		30:
			ActualResult := TestFBBusy.Busy;
			AssertEquals_BOOL(Expected := ExpectedResult, Actual := ActualResult, Message := 'Function Block was not busy when Extending');
			TEST_FINISHED();
			State := State + 10;
	END_CASE

	//Call to FB Cyclic Logic
	TestFBBusy.CyclicLogic();
END_IF
END_METHOD

METHOD CommandInhibited
VAR_INST
	State		   : INT;
	ActualResult   : BOOL;
	ExpectedResult : BOOL := TRUE;
END_VAR
IF TEST_ORDERED('CommandInhibitedAlarm') THEN
	CASE State OF
		0:
			IF TestFBAlarm15.InitComplete THEN
				TestFBAlarm15.Override := 0;
				TestFBAlarm15.MoveAbsolute(100, TRUE);
				State := State + 10;
			END_IF

		10:
			IF TestFBAlarm15.Error OR (TestFBAlarm15.InPosition AND NOT TestFBAlarm15.Busy) THEN
				ActualResult := TestFBAlarm15.BasicAxisAlarms[E_BasicAxis.CommandWhileInhibited].bRaised;
				State		 := State + 10;
			END_IF

		20:
			AssertEquals_BOOL(Expected := ExpectedResult, Actual := ActualResult, Message := 'The alarm was not raised for Command Inhibited Error');
			TEST_FINISHED();
			State := State + 10;
	END_CASE

	TestFBAlarm15.CyclicLogic();
END_IF
END_METHOD

METHOD Init
VAR_INST
	State		   : INT;
	ActualResult   : BOOL;
	ExpectedResult : BOOL := TRUE;
	Timeout		   : TON;
END_VAR
IF TEST_ORDERED('BasicAxisInit') THEN
	CASE State OF
		0:
			Timeout.IN := TRUE;
			State	   := State + 10;

		10:
			IF TestFBInit.InitComplete AND NOT TestFBInit.Busy THEN
				State := State + 10;
			END_IF

			IF Timeout.Q THEN
				State := State + 10;
			END_IF

		20:
			ActualResult := TestFBInit.InitComplete;
			AssertEquals_BOOL(Expected := ExpectedResult, Actual := ActualResult, Message := 'Function Block did not init complete in 2s');
			TEST_FINISHED();
			State := State + 10;
	END_CASE

	//Call to FB Cyclic Logic
	Timeout(PT := T#2S);
	TestFBInit.CyclicLogic();
END_IF
END_METHOD

METHOD MCHaltAlarm
VAR_INST
	State		   : INT;
	ActualResult   : BOOL;
	ExpectedResult : BOOL := TRUE;
	WriteADS	   : FB_WriteAdsSymByName;
END_VAR
IF TEST_ORDERED('MCHaltAlarm') THEN
	CASE State OF
		0:
			WriteADS(bWrite	  := TRUE,
					 sNetId	  := '',
					 nPort	  := 851,
					 sVarName := 'PRG_TEST.ComponentBasicAxisTest.TestFBAlarm4.BasicAxis.MCHalt.Error',
					 nSrcAddr := ADR(ExpectedResult),
					 nLen	  := SIZEOF(ExpectedResult),
					 tTimeout := T#2S,
					 eComMode :=,
					 bBusy	  =>,
					 bError	  =>,
					 nErrorId =>);

			IF NOT WriteADS.bBusy OR WriteADS.bError THEN
				State := State + 10;
			END_IF

			IF TestFBAlarm4.BasicAxisAlarms[E_BasicAxis.HaltError].bRaised THEN
				ActualResult := TestFBAlarm4.BasicAxisAlarms[E_BasicAxis.HaltError].bRaised;
				State		 := State + 10;
			END_IF

		10:
			AssertEquals_BOOL(Expected := ExpectedResult, Actual := ActualResult, Message := 'The alarm was not raised for MC_Halt.Error');
			TEST_FINISHED();
			State := State + 10;
	END_CASE

	TestFBAlarm4.CyclicLogic();
END_IF
END_METHOD

METHOD MCHomeAlarm
VAR_INST
	State		   : INT;
	ActualResult   : BOOL;
	ExpectedResult : BOOL := TRUE;
	WriteADS	   : FB_WriteAdsSymByName;
END_VAR
IF TEST_ORDERED('MCHomeAlarm') THEN
	CASE State OF
		0:
			WriteADS(bWrite	  := TRUE,
					 sNetId	  := '',
					 nPort	  := 851,
					 sVarName := 'PRG_TEST.ComponentBasicAxisTest.TestFBAlarm6.BasicAxis.DefaultHome._Error',
					 nSrcAddr := ADR(ExpectedResult),
					 nLen	  := SIZEOF(ExpectedResult),
					 tTimeout := T#2S,
					 eComMode :=,
					 bBusy	  =>,
					 bError	  =>,
					 nErrorId =>);

			IF NOT WriteADS.bBusy OR WriteADS.bError THEN
				State := State + 10;
			END_IF

			IF TestFBAlarm6.BasicAxisAlarms[E_BasicAxis.HomeError].bRaised THEN
				ActualResult := TestFBAlarm6.BasicAxisAlarms[E_BasicAxis.HomeError].bRaised;
				State		 := State + 10;
			END_IF

		10:
			AssertEquals_BOOL(Expected := ExpectedResult, Actual := ActualResult, Message := 'The alarm was not raised for HomeMethod.Error');
			TEST_FINISHED();
			State := State + 10;
	END_CASE

	TestFBAlarm6.CyclicLogic();
END_IF
END_METHOD

METHOD MCJogAlarm
VAR_INST
	State		   : INT;
	ActualResult   : BOOL;
	ExpectedResult : BOOL := TRUE;
	WriteADS	   : FB_WriteAdsSymByName;
END_VAR
IF TEST_ORDERED('MCJogAlarm') THEN
	CASE State OF
		0:
			WriteADS(bWrite	  := TRUE,
					 sNetId	  := '',
					 nPort	  := 851,
					 sVarName := 'PRG_TEST.ComponentBasicAxisTest.TestFBAlarm7.BasicAxis.MCJog.Error',
					 nSrcAddr := ADR(ExpectedResult),
					 nLen	  := SIZEOF(ExpectedResult),
					 tTimeout := T#2S,
					 eComMode :=,
					 bBusy	  =>,
					 bError	  =>,
					 nErrorId =>);

			IF NOT WriteADS.bBusy OR WriteADS.bError THEN
				State := State + 10;
			END_IF

			IF TestFBAlarm7.BasicAxisAlarms[E_BasicAxis.JogError].bRaised THEN
				ActualResult := TestFBAlarm7.BasicAxisAlarms[E_BasicAxis.JogError].bRaised;
				State		 := State + 10;
			END_IF

		10:
			AssertEquals_BOOL(Expected := ExpectedResult, Actual := ActualResult, Message := 'The alarm was not raised for MCJog.Error');
			TEST_FINISHED();
			State := State + 10;
	END_CASE

	TestFBAlarm7.CyclicLogic();
END_IF
END_METHOD

METHOD MCMoveAbsoluteAlarm
VAR_INST
	State		   : INT;
	ActualResult   : BOOL;
	ExpectedResult : BOOL := TRUE;
END_VAR
IF TEST_ORDERED('MCMoveAbsAlarm') THEN
	CASE State OF
		0:
			IF TestFBAlarm8.InitComplete THEN
				TestFBAlarm8.MoveAbsolute(100, TRUE);
				State := State + 10;
			END_IF

		10:
			IF TestFBAlarm8.Error OR (TestFBAlarm8.InPosition AND NOT TestFBAlarm8.Busy) THEN
				State := State + 10;
			END_IF

		20:
			ActualResult := TestFBAlarm8.BasicAxisAlarms[E_BasicAxis.MoveAbsoluteError].bRaised;
			AssertEquals_BOOL(Expected := ExpectedResult, Actual := ActualResult, Message := 'The alarm was not raised for Move Absolute Error');
			TEST_FINISHED();
			State := State + 10;
	END_CASE

	TestFBAlarm8.CyclicLogic();
END_IF
END_METHOD

METHOD MCMoveModulo
VAR_INST
	State		   : INT;
	ActualResult   : BOOL;
	ExpectedResult : BOOL := TRUE;
END_VAR
IF TEST_ORDERED('MCMoveModuloAlarm') THEN
	CASE State OF
		0:
			IF TestFBAlarm11.InitComplete THEN
				TestFBAlarm11.MoveModulo(100, MC_Direction.MC_Positive_Direction, TRUE);
				State := State + 10;
			END_IF

		10:
			IF TestFBAlarm11.Error OR (TestFBAlarm11.InPosition AND NOT TestFBAlarm11.Busy) THEN
				State := State + 10;
			END_IF

		20:
			ActualResult := TestFBAlarm11.BasicAxisAlarms[E_BasicAxis.MoveModuloError].bRaised;
			AssertEquals_BOOL(Expected := ExpectedResult, Actual := ActualResult, Message := 'The alarm was not raised for Move Modulo Error');
			TEST_FINISHED();
			State := State + 10;
	END_CASE

	TestFBAlarm11.CyclicLogic();
END_IF
END_METHOD

METHOD MCMoveRelativeAlarm
VAR_INST
	State		   : INT;
	ActualResult   : BOOL;
	ExpectedResult : BOOL := TRUE;
END_VAR
IF TEST_ORDERED('MCMoveAbsAlarm') THEN
	CASE State OF
		0:
			IF TestFBAlarm9.InitComplete THEN
				TestFBAlarm9.MoveRelative(100, TRUE);
				State := State + 10;
			END_IF

		10:
			IF TestFBAlarm9.Error OR (TestFBAlarm9.InPosition AND NOT TestFBAlarm9.Busy) THEN
				State := State + 10;
			END_IF

		20:
			ActualResult := TestFBAlarm9.BasicAxisAlarms[E_BasicAxis.MoveRelativeError].bRaised;
			AssertEquals_BOOL(Expected := ExpectedResult, Actual := ActualResult, Message := 'The alarm was not raised for Move Relative Error');
			TEST_FINISHED();
			State := State + 10;
	END_CASE

	TestFBAlarm9.CyclicLogic();
END_IF
END_METHOD

METHOD MCMoveVelocity
VAR_INST
	State		   : INT;
	ActualResult   : BOOL;
	ExpectedResult : BOOL := TRUE;
END_VAR
IF TEST_ORDERED('MCMoveVelAlarm') THEN
	CASE State OF
		0:
			IF TestFBAlarm10.InitComplete THEN
				TestFBAlarm10.MoveVelocity(100, TRUE);
				State := State + 10;
			END_IF

		10:
			IF TestFBAlarm10.Error OR (TestFBAlarm10.InPosition AND NOT TestFBAlarm10.Busy) THEN
				State := State + 10;
			END_IF

		20:
			ActualResult := TestFBAlarm10.BasicAxisAlarms[E_BasicAxis.MoveVelocityError].bRaised;
			AssertEquals_BOOL(Expected := ExpectedResult, Actual := ActualResult, Message := 'The alarm was not raised for Move Relative Error');
			TEST_FINISHED();
			State := State + 10;
	END_CASE

	TestFBAlarm10.CyclicLogic();
END_IF
END_METHOD

METHOD MCPowerAlarm
VAR_INST
	State		   : INT;
	ActualResult   : BOOL;
	ExpectedResult : BOOL := TRUE;
	WriteADS	   : FB_WriteAdsSymByName;
END_VAR
IF TEST_ORDERED('MCPowerAlarm') THEN
	CASE State OF
		0:
			WriteADS(bWrite	  := TRUE,
					 sNetId	  := '',
					 nPort	  := 851,
					 sVarName := 'PRG_TEST.ComponentBasicAxisTest.TestFBAlarm2.BasicAxis.MCPower.Error',
					 nSrcAddr := ADR(ExpectedResult),
					 nLen	  := SIZEOF(ExpectedResult),
					 tTimeout := T#2S,
					 eComMode :=,
					 bBusy	  =>,
					 bError	  =>,
					 nErrorId =>);

			IF NOT WriteADS.bBusy OR WriteADS.bError THEN
				State := State + 10;
			END_IF

			IF TestFBAlarm2.BasicAxisAlarms[E_BasicAxis.PowerError].bRaised THEN
				ActualResult := TestFBAlarm2.BasicAxisAlarms[E_BasicAxis.PowerError].bRaised;
				State		 := State + 10;
			END_IF

		10:
			AssertEquals_BOOL(Expected := ExpectedResult, Actual := ActualResult, Message := 'The alarm was not raised for MC_Power.Error');
			TEST_FINISHED();
			State := State + 10;
	END_CASE

	TestFBAlarm2.CyclicLogic();
END_IF
END_METHOD

METHOD McReadAxisParametersAlarm
VAR_INST
	State		   : INT;
	ActualResult   : BOOL;
	ExpectedResult : BOOL := TRUE;
	WriteADS	   : FB_WriteAdsSymByName;
END_VAR
IF TEST_ORDERED('MCReadAxisAlarm') THEN
	CASE State OF
		0:
			WriteADS(bWrite	  := TRUE,
					 sNetId	  := '',
					 nPort	  := 851,
					 sVarName := 'PRG_TEST.ComponentBasicAxisTest.TestFBAlarm12.BasicAxis.MCReadParameterSet.Error',
					 nSrcAddr := ADR(ExpectedResult),
					 nLen	  := SIZEOF(ExpectedResult),
					 tTimeout := T#2S,
					 eComMode :=,
					 bBusy	  =>,
					 bError	  =>,
					 nErrorId =>);

			IF NOT WriteADS.bBusy OR WriteADS.bError THEN
				State := State + 10;
			END_IF

			IF TestFBAlarm12.BasicAxisAlarms[E_BasicAxis.ReadParameterSetError].bRaised THEN
				ActualResult := TestFBAlarm12.BasicAxisAlarms[E_BasicAxis.ReadParameterSetError].bRaised;
				State		 := State + 10;
			END_IF

		10:
			AssertEquals_BOOL(Expected := ExpectedResult, Actual := ActualResult, Message := 'The alarm was not raised for MC Read Axis Parameter Error');
			TEST_FINISHED();
			State := State + 10;
	END_CASE

	TestFBAlarm12.CyclicLogic();
END_IF
END_METHOD

METHOD MCResetAlarm
VAR_INST
	State		   : INT;
	ActualResult   : BOOL;
	ExpectedResult : BOOL := TRUE;
	WriteADS	   : FB_WriteAdsSymByName;
END_VAR
IF TEST_ORDERED('MCResetAlarm') THEN
	CASE State OF
		0:
			WriteADS(bWrite	  := TRUE,
					 sNetId	  := '',
					 nPort	  := 851,
					 sVarName := 'PRG_TEST.ComponentBasicAxisTest.TestFBAlarm3.BasicAxis.DefaultReset._Error',
					 nSrcAddr := ADR(ExpectedResult),
					 nLen	  := SIZEOF(ExpectedResult),
					 tTimeout := T#2S,
					 eComMode :=,
					 bBusy	  =>,
					 bError	  =>,
					 nErrorId =>);

			IF NOT WriteADS.bBusy OR WriteADS.bError THEN
				State := State + 10;
			END_IF

			IF TestFBAlarm3.BasicAxisAlarms[E_BasicAxis.ResetError].bRaised THEN
				ActualResult := TestFBAlarm3.BasicAxisAlarms[E_BasicAxis.ResetError].bRaised;
				State		 := State + 10;
			END_IF

		10:
			AssertEquals_BOOL(Expected := ExpectedResult, Actual := ActualResult, Message := 'The alarm was not raised for ResetMethod.Error');
			TEST_FINISHED();
			State := State + 10;
	END_CASE

	TestFBAlarm3.CyclicLogic();
END_IF
END_METHOD

METHOD McWriteAxisBoolParameterAlarm
VAR_INST
	State		   : INT;
	ActualResult   : BOOL;
	ExpectedResult : BOOL := TRUE;
	WriteADS	   : FB_WriteAdsSymByName;
END_VAR
IF TEST_ORDERED('MCWriteAxisBoolAlarm') THEN
	CASE State OF
		0:
			WriteADS(bWrite	  := TRUE,
					 sNetId	  := '',
					 nPort	  := 851,
					 sVarName := 'PRG_TEST.ComponentBasicAxisTest.TestFBAlarm14.BasicAxis.MCWriteBoolParameter.Error',
					 nSrcAddr := ADR(ExpectedResult),
					 nLen	  := SIZEOF(ExpectedResult),
					 tTimeout := T#2S,
					 eComMode :=,
					 bBusy	  =>,
					 bError	  =>,
					 nErrorId =>);

			IF NOT WriteADS.bBusy OR WriteADS.bError THEN
				State := State + 10;
			END_IF

			IF TestFBAlarm14.BasicAxisAlarms[E_BasicAxis.WriteBoolParameterError].bRaised THEN
				ActualResult := TestFBAlarm14.BasicAxisAlarms[E_BasicAxis.WriteBoolParameterError].bRaised;
				State		 := State + 10;
			END_IF

		10:
			AssertEquals_BOOL(Expected := ExpectedResult, Actual := ActualResult, Message := 'The alarm was not raised for MC Write Axis Bool Parameter Error');
			TEST_FINISHED();
			State := State + 10;
	END_CASE

	TestFBAlarm14.CyclicLogic();
END_IF
END_METHOD

METHOD McWriteAxisParameterAlarm
VAR_INST
	State		   : INT;
	ActualResult   : BOOL;
	ExpectedResult : BOOL := TRUE;
	WriteADS	   : FB_WriteAdsSymByName;
END_VAR
IF TEST_ORDERED('MCWriteAxisAlarm') THEN
	CASE State OF
		0:
			WriteADS(bWrite	  := TRUE,
					 sNetId	  := '',
					 nPort	  := 851,
					 sVarName := 'PRG_TEST.ComponentBasicAxisTest.TestFBAlarm13.BasicAxis.MCWriteParameter.Error',
					 nSrcAddr := ADR(ExpectedResult),
					 nLen	  := SIZEOF(ExpectedResult),
					 tTimeout := T#2S,
					 eComMode :=,
					 bBusy	  =>,
					 bError	  =>,
					 nErrorId =>);

			IF NOT WriteADS.bBusy OR WriteADS.bError THEN
				State := State + 10;
			END_IF

			IF TestFBAlarm13.BasicAxisAlarms[E_BasicAxis.WriteParameterError].bRaised THEN
				ActualResult := TestFBAlarm13.BasicAxisAlarms[E_BasicAxis.WriteParameterError].bRaised;
				State		 := State + 10;
			END_IF

		10:
			AssertEquals_BOOL(Expected := ExpectedResult, Actual := ActualResult, Message := 'The alarm was not raised for MC Write Axis Parameter Error');
			TEST_FINISHED();
			State := State + 10;
	END_CASE

	TestFBAlarm13.CyclicLogic();
END_IF
END_METHOD

METHOD NameSetProperty
VAR_INST
	State			: INT;
	ActualResult	: STRING;
	ActualResultHMI : STRING;
	ExpectedResult	: STRING := 'TEST_NAME';
END_VAR
IF TEST_ORDERED('BasicAxisNameSetProperty') THEN
	CASE State OF
		0:
			State := State + 10;

		10:
			IF TestFBNameSetProperty.InitComplete AND NOT TestFBNameSetProperty.Busy THEN
				State := State + 10;
			END_IF

		20:
			TestFBNameSetProperty.Name := ExpectedResult;
			State					   := State + 10;

		30:
			ActualResultHMI := TestFBNameSetProperty.ComponentBase_HMI.Config.Name;
			ActualResult	:= TestFBNameSetProperty.Name;
			AssertEquals(Expected := ExpectedResult, Actual := ActualResult, Message := 'Name was not read by Property correctly');
			AssertEquals(Expected := ExpectedResult, Actual := ActualResultHMI, Message := 'Name was not read by HMI correctly');
			TEST_FINISHED();
			State := State + 10;
	END_CASE

	//Call to FB Cyclic Logic
	TestFBNameSetProperty.CyclicLogic();
END_IF
END_METHOD

METHOD SimulationCheckAlarm
VAR_INST
	State		   : INT;
	ActualResult   : BOOL;
	ExpectedResult : BOOL := TRUE;
END_VAR
IF TEST_ORDERED('BasicAxisSimulationCheckAlarm') THEN
	CASE State OF
		0:
			State := State + 10;

		10:
			IF TestFBSimulationCheckAlarm.InitComplete AND NOT TestFBSimulationCheckAlarm.Busy THEN
				State := State + 10;
			END_IF

		20:
			TestFBSimulationCheckAlarm.InSimulation := TRUE; //Set simulation to true;
			State									:= State + 10;

		30:
			ActualResult := TestFBSimulationCheckAlarm.ComponentBaseAlarms[E_ComponentBase.SimulationWarning].bRaised;
			AssertEquals_BOOL(Expected := ExpectedResult, Actual := ActualResult, Message := 'Function Block did Raise alarm when in simulation');
			TEST_FINISHED();
			State := State + 10;
	END_CASE

	//Call to FB Cyclic Logic
	TestFBSimulationCheckAlarm.CyclicLogic();
END_IF
END_METHOD

METHOD SimulationSetHMI
VAR_INST
	State			: INT;
	ActualResult	: BOOL;
	ActualResultHMI : BOOL;
	ExpectedResult	: BOOL := TRUE;
	WriteADS		: FB_WriteAdsSymByName;
END_VAR
IF TEST_ORDERED('BasicAxisSetSimulationHMI') THEN
	CASE State OF
		0:
			State := State + 10;

		10:
			IF TestFBSimulationSetHMI.InitComplete AND NOT TestFBSimulationSetHMI.Busy THEN
				TestFBSimulationSetHMI.AllowHMIControl(); // Must turn on Allow control for code to function
				State := State + 10;
			END_IF

		20:
			WriteADS(bWrite	  := TRUE,
					 sNetId	  := '',
					 nPort	  := 851,
					 sVarName := 'PRG_TEST.ComponentBasicAxisTest.TestFBSimulationSetHMI.ComponentBase_HMI.Command.SimulatedOperation',
					 nSrcAddr := ADR(ExpectedResult),
					 nLen	  := SIZEOF(ExpectedResult),
					 tTimeout := T#2S,
					 eComMode :=,
					 bBusy	  =>,
					 bError	  =>,
					 nErrorId =>);

			IF NOT WriteADS.bBusy OR WriteADS.bError THEN
				State := State + 10;
			END_IF

		30:
			ActualResult	:= TestFBSimulationSetHMI.InSimulation;
			ActualResultHMI := TestFBSimulationSetHMI.ComponentBase_HMI.Status.InSimulation;
			AssertEquals_BOOL(Expected := ExpectedResult, Actual := ActualResult, Message := 'Function Block did not set simulation by HMI when read by Property');
			AssertEquals_BOOL(Expected := ExpectedResult, Actual := ActualResultHMI, Message := 'Function Block did not set simulation by HMI when read by HMI');
			TEST_FINISHED();
			State := State + 10;
	END_CASE

	//Call to FB Cyclic Logic
	TestFBSimulationSetHMI.CyclicLogic();
END_IF
END_METHOD

METHOD SimulationSetProperty
VAR_INST
	State			: INT;
	ActualResult	: BOOL;
	ActualResultHMI : BOOL;
	ExpectedResult	: BOOL := TRUE;
END_VAR
IF TEST_ORDERED('BasicAxisSetSimulationProperty') THEN
	CASE State OF
		0:
			State := State + 10;

		10:
			IF TestFBSimulationSetProperty.InitComplete AND NOT TestFBSimulationSetProperty.Busy THEN
				State := State + 10;
			END_IF

		20:
			TestFBSimulationSetProperty.InSimulation := TRUE;
			State									 := State + 10;

		30:
			ActualResult	:= TestFBSimulationSetProperty.InSimulation;
			ActualResultHMI := TestFBSimulationSetProperty.ComponentBase_HMI.Status.InSimulation;
			AssertEquals_BOOL(Expected := ExpectedResult, Actual := ActualResult, Message := 'Function Block did not set simulation by property when read by Property');
			AssertEquals_BOOL(Expected := ExpectedResult, Actual := ActualResultHMI, Message := 'Function Block did not set simulation by property when read by HMI');
			TEST_FINISHED();
			State := State + 10;
	END_CASE

	//Call to FB Cyclic Logic
	TestFBSimulationSetProperty.CyclicLogic();
END_IF
END_METHOD

END_FUNCTION_BLOCK

// Testing/PRG_TEST
PROGRAM PRG_TEST
VAR
	SingleSolenoidTest		   : FB_SingleSolenoid_Test;
	DoubleSolenoidTest		   : FB_DoubleSolenoid_Test;
	SingleSolenoidFeedbackTest : FB_SingleSolenoidFeedback_Test;
	ComponentBasicAxisTest	   : FB_ComponentBasicAxis_Test;
END_VAR

TcUnit.RUN();

END_PROGRAM

// Testing/Solenoids/FB_SingleSolenoid_Test
FUNCTION_BLOCK FB_SingleSolenoid_Test EXTENDS TcUnit.FB_TestSuite
VAR
	// FBs for ComponentBase
	TestFBInit					: FB_SingleSolenoid;
	TestFBNameSetProperty		: FB_SingleSolenoid;
	TestFBNameSetHMI			: FB_SingleSolenoid;
	TestFBSimulationSetProperty : FB_SingleSolenoid;
	TestFBSimulationSetHMI		: FB_SingleSolenoid;
	TestFBSimulationCheckAlarm	: FB_SingleSolenoid;
	TestFBBusy					: FB_SingleSolenoid;
	TestFBAllowHMI				: FB_SingleSolenoid;
	TestFBBlockHMI				: FB_SingleSolenoid;

	// Solenoid FB	
	TestSingleSolenoidExtend  : FB_SingleSolenoid;
	TestSingleSolenoidRetract : FB_SingleSolenoid;
END_VAR

Init();
NameSetProperty();
SimulationSetProperty();
SimulationSetHMI();
SimulationCheckAlarm();
Busy();
AllowHMI();
BlockHMI();
ExtendEqualsExtendedOutputOn();
RetractEqualsExtendOutputOff();

METHOD AllowHMI
VAR_INST
	State		   : INT;
	ActualResult   : BOOL;
	ExpectedResult : BOOL := TRUE;
END_VAR
IF TEST_ORDERED('AllowHMI') THEN
	CASE State OF
		0:
			State := State + 10;

		10:
			IF TestFBAllowHMI.InitComplete AND NOT TestFBAllowHMI.Busy THEN
				TestFBAllowHMI.AllowHMIControl();
				State := State + 10;
			END_IF

		20:
			ActualResult := TestFBAllowHMI.ComponentBase_HMI.Status.HMIControlAvailable;
			AssertEquals_BOOL(Expected := ExpectedResult, Actual := ActualResult, Message := 'Function Block read allow HMI Control in HMI Tag not true');
			TEST_FINISHED();
			State := State + 10;
	END_CASE

	//Call to FB Cyclic Logic
	TestFBAllowHMI.CyclicLogic();
END_IF
END_METHOD

METHOD BlockHMI
VAR_INST
	State		   : INT;
	ActualResult   : BOOL;
	ExpectedResult : BOOL := FALSE;
END_VAR
IF TEST_ORDERED('BlockHMI') THEN
	CASE State OF
		0:
			State := State + 10;

		10:
			IF TestFBBlockHMI.InitComplete AND NOT TestFBBlockHMI.Busy THEN
				TestFBBlockHMI.AllowHMIControl();
				State := State + 10;
			END_IF

		20:
			IF TestFBBlockHMI.ComponentBase_HMI.Status.HMIControlAvailable THEN
				TestFBBlockHMI.BlockHMIControl();
				State := State + 10;
			END_IF

		30:
			ActualResult := TestFBBlockHMI.ComponentBase_HMI.Status.HMIControlAvailable;
			AssertEquals_BOOL(Expected := ExpectedResult, Actual := ActualResult, Message := 'Function Block read Block HMI Control in HMI Tag not false');
			TEST_FINISHED();
			State := State + 10;
	END_CASE

	//Call to FB Cyclic Logic
	TestFBBlockHMI.CyclicLogic();
END_IF
END_METHOD

METHOD Busy
VAR_INST
	State		   : INT;
	ActualResult   : BOOL;
	ExpectedResult : BOOL := TRUE;
	Timeout		   : TON;
END_VAR
IF TEST_ORDERED('Busy') THEN
	CASE State OF
		0:
			State := State + 10;

		10:
			IF TestFBBusy.InitComplete AND NOT TestFBBusy.Busy THEN
				State := State + 10;
			END_IF

		20:
			TestFBBusy.Extend();
			State := State + 10;

		30:
			ActualResult := TestFBBusy.Busy;
			AssertEquals_BOOL(Expected := ExpectedResult, Actual := ActualResult, Message := 'Function Block was not busy when Extending');
			TEST_FINISHED();
			State := State + 10;
	END_CASE

	//Call to FB Cyclic Logic
	TestFBBusy.CyclicLogic();
END_IF
END_METHOD

METHOD ExtendEqualsExtendedOutputOn
VAR_INST
	State		   : INT;
	ActualResult   : BOOL;
	ExpectedResult : BOOL := TRUE;
END_VAR
IF TEST_ORDERED('ExtendEqualsExtendedOutputOn') THEN
	CASE State OF
		0:
			State := State + 10;

		10:
			TestSingleSolenoidExtend.Extend();
			State := State + 10;

		20:
			ActualResult := TestSingleSolenoidExtend.ExtendOutput;
			AssertEquals_BOOL(Expected := ExpectedResult, Actual := ActualResult, Message := 'Solenoid did not set output on');
			TEST_FINISHED();
			State := State + 10;
	END_CASE

	TestSingleSolenoidExtend.CyclicLogic();
END_IF
END_METHOD

METHOD Init
VAR_INST
	State		   : INT;
	ActualResult   : BOOL;
	ExpectedResult : BOOL := TRUE;
	Timeout		   : TON;
END_VAR
IF TEST_ORDERED('Init') THEN
	CASE State OF
		0:
			Timeout.IN := TRUE;
			State	   := State + 10;

		10:
			IF TestFBInit.InitComplete AND NOT TestFBInit.Busy THEN
				State := State + 10;
			END_IF

			IF Timeout.Q THEN
				State := State + 10;
			END_IF

		20:
			ActualResult := TestFBInit.InitComplete;
			AssertEquals_BOOL(Expected := ExpectedResult, Actual := ActualResult, Message := 'Function Block did not init complete in 2s');
			TEST_FINISHED();
			State := State + 10;
	END_CASE

	//Call to FB Cyclic Logic
	Timeout(PT := T#2S);
	TestFBInit.CyclicLogic();
END_IF
END_METHOD

METHOD NameSetProperty
VAR_INST
	State			: INT;
	ActualResult	: STRING;
	ActualResultHMI : STRING;
	ExpectedResult	: STRING := 'TEST_NAME';
END_VAR
IF TEST_ORDERED('NameSetProperty') THEN
	CASE State OF
		0:
			State := State + 10;

		10:
			IF TestFBNameSetProperty.InitComplete AND NOT TestFBNameSetProperty.Busy THEN
				State := State + 10;
			END_IF

		20:
			TestFBNameSetProperty.Name := ExpectedResult;
			State					   := State + 10;

		30:
			ActualResultHMI := TestFBNameSetProperty.ComponentBase_HMI.Config.Name;
			ActualResult	:= TestFBNameSetProperty.Name;
			AssertEquals(Expected := ExpectedResult, Actual := ActualResult, Message := 'Name was not read by Property correctly');
			AssertEquals(Expected := ExpectedResult, Actual := ActualResultHMI, Message := 'Name was not read by HMI correctly');
			TEST_FINISHED();
			State := State + 10;
	END_CASE

	//Call to FB Cyclic Logic
	TestFBNameSetProperty.CyclicLogic();
END_IF
END_METHOD

METHOD RetractEqualsExtendOutputOff
VAR_INST
	State		   : INT;
	ActualResult   : BOOL;
	ExpectedResult : BOOL := FALSE;
END_VAR
IF TEST_ORDERED('RetractEqualsExtendOutputOff') THEN
	CASE State OF
		0:
			State := State + 10;

		10:
			TestSingleSolenoidRetract.Retract();
			State := State + 10;

		20:
			ActualResult := TestSingleSolenoidRetract.ExtendOutput;
			AssertEquals_BOOL(Expected := ExpectedResult, Actual := ActualResult, Message := 'Solenoid did not set output on');
			TEST_FINISHED();
			State := State + 10;
	END_CASE

	TestSingleSolenoidRetract.CyclicLogic();
END_IF
END_METHOD

METHOD SimulationCheckAlarm
VAR_INST
	State		   : INT;
	ActualResult   : BOOL;
	ExpectedResult : BOOL := TRUE;
END_VAR
IF TEST_ORDERED('SimulationCheckAlarm') THEN
	CASE State OF
		0:
			State := State + 10;

		10:
			IF TestFBSimulationCheckAlarm.InitComplete AND NOT TestFBSimulationCheckAlarm.Busy THEN
				State := State + 10;
			END_IF

		20:
			TestFBSimulationCheckAlarm.InSimulation := TRUE; //Set simulation to true;
			State									:= State + 10;

		30:
			ActualResult := TestFBSimulationCheckAlarm.ComponentBaseAlarms[E_ComponentBase.SimulationWarning].bRaised;
			AssertEquals_BOOL(Expected := ExpectedResult, Actual := ActualResult, Message := 'Function Block did Raise alarm when in simulation');
			TEST_FINISHED();
			State := State + 10;
	END_CASE

	//Call to FB Cyclic Logic
	TestFBSimulationCheckAlarm.CyclicLogic();
END_IF
END_METHOD

METHOD SimulationSetHMI
VAR_INST
	State			: INT;
	ActualResult	: BOOL;
	ActualResultHMI : BOOL;
	ExpectedResult	: BOOL := TRUE;
	WriteADS		: FB_WriteAdsSymByName;
END_VAR
IF TEST_ORDERED('SimulationSetHMI') THEN
	CASE State OF
		0:
			State := State + 10;

		10:
			IF TestFBSimulationSetHMI.InitComplete AND NOT TestFBSimulationSetHMI.Busy THEN
				TestFBSimulationSetHMI.AllowHMIControl(); // Must turn on Allow control for code to function
				State := State + 10;
			END_IF

		20:
			WriteADS(bWrite	  := TRUE,
					 sNetId	  := '',
					 nPort	  := 851,
					 sVarName := 'PRG_TEST.SingleSolenoidTest.TestFBSimulationSetHMI.ComponentBase_HMI.Command.SimulatedOperation',
					 nSrcAddr := ADR(ExpectedResult),
					 nLen	  := SIZEOF(ExpectedResult),
					 tTimeout := T#2S,
					 eComMode :=,
					 bBusy	  =>,
					 bError	  =>,
					 nErrorId =>);

			IF NOT WriteADS.bBusy OR WriteADS.bError THEN
				State := State + 10;
			END_IF

		30:
			ActualResult	:= TestFBSimulationSetHMI.InSimulation;
			ActualResultHMI := TestFBSimulationSetHMI.ComponentBase_HMI.Status.InSimulation;
			AssertEquals_BOOL(Expected := ExpectedResult, Actual := ActualResult, Message := 'Function Block did not set simulation by HMI when read by Property');
			AssertEquals_BOOL(Expected := ExpectedResult, Actual := ActualResultHMI, Message := 'Function Block did not set simulation by HMI when read by HMI');
			TEST_FINISHED();
			State := State + 10;
	END_CASE

	//Call to FB Cyclic Logic
	TestFBSimulationSetHMI.CyclicLogic();
END_IF
END_METHOD

METHOD SimulationSetProperty
VAR_INST
	State			: INT;
	ActualResult	: BOOL;
	ActualResultHMI : BOOL;
	ExpectedResult	: BOOL := TRUE;
END_VAR
IF TEST_ORDERED('SimulationSetProperty') THEN
	CASE State OF
		0:
			State := State + 10;

		10:
			IF TestFBSimulationSetProperty.InitComplete AND NOT TestFBSimulationSetProperty.Busy THEN
				State := State + 10;
			END_IF

		20:
			TestFBSimulationSetProperty.InSimulation := TRUE;
			State									 := State + 10;

		30:
			ActualResult	:= TestFBSimulationSetProperty.InSimulation;
			ActualResultHMI := TestFBSimulationSetProperty.ComponentBase_HMI.Status.InSimulation;
			AssertEquals_BOOL(Expected := ExpectedResult, Actual := ActualResult, Message := 'Function Block did not set simulation by property when read by Property');
			AssertEquals_BOOL(Expected := ExpectedResult, Actual := ActualResultHMI, Message := 'Function Block did not set simulation by property when read by HMI');
			TEST_FINISHED();
			State := State + 10;
	END_CASE

	//Call to FB Cyclic Logic
	TestFBSimulationSetProperty.CyclicLogic();
END_IF
END_METHOD

END_FUNCTION_BLOCK

// Testing/Solenoids/FB_DoubleSolenoid_Test
FUNCTION_BLOCK FB_DoubleSolenoid_Test EXTENDS TcUnit.FB_TestSuite
VAR
	TestFBExtend  : FB_DoubleSolenoid;
	TestFBRetract : FB_DoubleSolenoid;
END_VAR

ExtendEqualsExtendOutputOnRetractOff();
RetractEqualsExtendOutputOffRetractOutputOn();

METHOD ExtendEqualsExtendOutputOnRetractOff
VAR_INST
	State						: INT;
	ActualExtendOutputResult	: BOOL;
	ActualRetractOutputResult	: BOOL;
	ExpectedExtendOutputResult	: BOOL := TRUE;
	ExpectedRetractOutputResult : BOOL := FALSE;
END_VAR
IF TEST_ORDERED('ExtendEqualsExtendOutputOnRetractOff') THEN
	CASE State OF
		0:
			State := State + 10;

		10:
			IF TestFBExtend.InitComplete AND NOT TestFBExtend.Busy THEN
				TestFBExtend.Extend();
				State := State + 10;
			END_IF

		20:
			ActualExtendOutputResult := TestFBExtend.ExtendOutput;
			AssertEquals_BOOL(Expected := ExpectedExtendOutputResult, Actual := ActualExtendOutputResult, Message := 'Solenoid did not set extend output on');
			ActualRetractOutputResult := TestFBExtend.RetractOutput;
			AssertEquals_BOOL(Expected := ExpectedRetractOutputResult, Actual := ActualRetractOutputResult, Message := 'Solenoid did not set retract output off');
			TEST_FINISHED();
			State := State + 10;
	END_CASE

	TestFBExtend.CyclicLogic();
END_IF
END_METHOD

METHOD RetractEqualsExtendOutputOffRetractOutputOn
VAR_INST
	State						: INT;
	ActualExtendOutputResult	: BOOL;
	ActualRetractOutputResult	: BOOL;
	ExpectedExtendOutputResult	: BOOL := FALSE;
	ExpectedRetractOutputResult : BOOL := TRUE;
END_VAR
IF TEST_ORDERED('ExtendEqualsExtendOutputOffRetractOn') THEN
	CASE State OF
		0:
			State := State + 10;

		10:
			IF TestFBRetract.InitComplete AND NOT TestFBRetract.Busy THEN
				TestFBRetract.Extend();
				State := State + 10;
			END_IF

		20:
			IF TestFBRetract.Extended THEN
				TestFBRetract.Retract();
				State := State + 10;
			END_IF

		30:
			ActualExtendOutputResult := TestFBRetract.ExtendOutput;
			AssertEquals_BOOL(Expected := ExpectedExtendOutputResult, Actual := ActualExtendOutputResult, Message := 'Solenoid did not set extend output off');
			ActualRetractOutputResult := TestFBRetract.RetractOutput;
			AssertEquals_BOOL(Expected := ExpectedRetractOutputResult, Actual := ActualRetractOutputResult, Message := 'Solenoid did not set retract output on');
			TEST_FINISHED();
			State := State + 10;
	END_CASE

	TestFBRetract.CyclicLogic();
END_IF
END_METHOD

END_FUNCTION_BLOCK

// Testing/Solenoids/FB_SingleSolenoidFeedback_Test
FUNCTION_BLOCK FB_SingleSolenoidFeedback_Test EXTENDS FB_TestSuite
VAR
	// Solenoid FB	
	TestSingleSolenoidFeedbackExtend	   : FB_SingleSolenoidFeedback;
	TestSingleSolenoidFeedbackExtendError  : FB_SingleSolenoidFeedback;
	TestSingleSolenoidFeedbackRetract	   : FB_SingleSolenoidFeedback;
	TestSingleSolenoidFeedbackRetractError : FB_SingleSolenoidFeedback;
END_VAR

Extend();
ExtendError();

METHOD Extend
VAR_INST
	State		   : INT;
	ActualResult   : BOOL;
	ExpectedResult : BOOL := TRUE;
END_VAR
IF TEST_ORDERED('SingleSolenoidFeedbackTestExtend') THEN
	CASE State OF
		0:
			IF TestSingleSolenoidFeedbackExtend.InitComplete AND NOT TestSingleSolenoidFeedbackExtend.Busy THEN
				TestSingleSolenoidFeedbackExtend.Extend();
				TestSingleSolenoidFeedbackExtend.ExtendedInput	:= TRUE;  //Set the feedback
				TestSingleSolenoidFeedbackExtend.RetractedInput := FALSE; //Set the feedback
				State											:= State + 10;
			END_IF

		10:
			ActualResult := TestSingleSolenoidFeedbackExtend.Extended;
			AssertEquals_BOOL(Expected := ExpectedResult, Actual := ActualResult, Message := 'Solenoid feedback did not turn on');
			State := State + 10;
			TEST_FINISHED();
	END_CASE

	TestSingleSolenoidFeedbackExtend.CyclicLogic();
END_IF
END_METHOD

METHOD ExtendError
VAR_INST
	State				: INT;
	ActualResult		: BOOL;
	ExpectedResult		: BOOL := FALSE;
	ActualErrorResult	: BOOL;
	ExpectedErrorResult : BOOL := TRUE;
END_VAR
IF TEST_ORDERED('SingleSolenoidFeedbackTestExtendError') THEN
	CASE State OF
		0:
			IF TestSingleSolenoidFeedbackExtendError.InitComplete AND NOT TestSingleSolenoidFeedbackExtendError.Busy THEN
				TestSingleSolenoidFeedbackExtendError.Extend();
				State := State + 10;
			END_IF

		10:
			IF TestSingleSolenoidFeedbackExtendError.Extended OR TestSingleSolenoidFeedbackExtendError.Error THEN
				ActualResult := TestSingleSolenoidFeedbackExtendError.Extended;
				AssertEquals_BOOL(Expected := ExpectedResult, Actual := ActualResult, Message := 'Solenoid feedback did not turn on');
				ActualErrorResult := TestSingleSolenoidFeedbackExtendError.Error;
				AssertEquals_BOOL(Expected := ExpectedErrorResult, Actual := ActualErrorResult, Message := 'Solenoid Feedback extend no error');
				State := State + 10;
				TEST_FINISHED();
			END_IF
	END_CASE

	TestSingleSolenoidFeedbackExtendError.CyclicLogic();
END_IF
END_METHOD

END_FUNCTION_BLOCK
